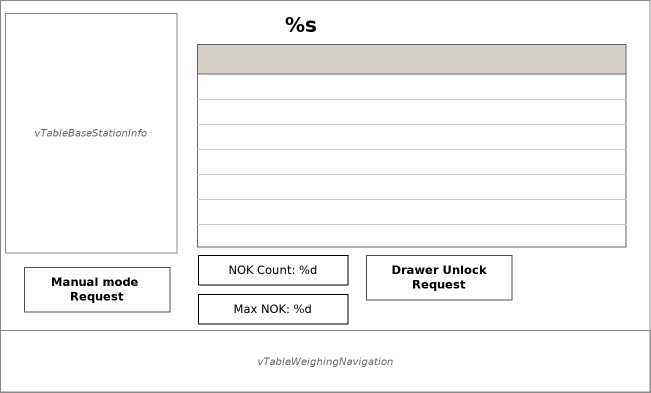
VISUALIZATION vTableWeighingDetail  // 651x393
VAR_IN_OUT
	fbStation:FB_WeighingStation;
	fbTableControl: FB_TableControl;
END_VAR
    Rectangle (0,0 650x392)
    Frame (5,13 172x240)
        shows vTableBaseStationInfo(fbStation := fbStation)
    Rectangle (226,10 150x30), "%s", text variable: fbStation.sStationName
    Table (197,44 429x203), data array: fbStation.fbTimeStats.astTT
        p3854506369: fbStation.fbTimeStats.astTT[INDEX].sStepName
        p1892666644: fbStation.fbTimeStats.astTT[INDEX].rStepTime
        p2232123230: Tests
        p1128707560: fbStation.fbTimeStats.uiTTLastIndex
    Frame (0,330 651x63)
        shows vTableWeighingNavigation(fbTableControl := fbTableControl)
    Rectangle (198,255 150x30), "NOK Count: %d", text variable: fbStation.stSettings.iNOK_BottleCounter
    Rectangle (198,294 150x30), "Max NOK: %d", text variable: fbStation.stSettings.iMaxNOK_Bottles
    Rectangle (366,255 146x45), "Drawer Unlock Request", colour toggle: fbStation.bDrawerUnlockRequest, input disabled if: fbStation.stSettings.iMaxNOK_Bottles = fbStation.stSettings.iNOK_BottleCounter
        toggle fbStation.bDrawerUnlockRequest
    Rectangle (24,267 146x45), "Manual mode Request", colour toggle: fbStation.bManualModeRequest
        toggle fbStation.bManualModeRequest
END_VISUALIZATION

(* stored: Version 1.1.0.1, ProductVersion 3.1.4024.15
   Visu vTableWeighingDetail: Id {f6cbcf01-8586-4561-a1dd-32a92e078c17} *)
